TYPE RefVector :
STRUCT
	input_len				: UDINT;
	hash					: STRING[262];
	keyed_hash				: STRING[262];
	derive_key				: STRING[262];
END_STRUCT
END_TYPE

(* stored: Version 1.1.0.1
   DUT RefVector: Id {bcf5e03d-1624-4151-874d-d0602a28fb27} *)
